Fanuc KAREL source: IO0221.KL

-- PROVISIONAL review KL for V1013-1; original PC SHA256 55de212278e1739486ba962373558651f202fb49e40d7032ca4ff645f1fc8ad3
-- Incomplete behavior may be omitted. Consult companion uncertainty JSON. Do not deploy.
PROGRAM IO0221
%NOLOCKGROUP
-- UNRESOLVED_LOCAL_POOL 5 cells at code offset 13; source declarations unknown
-- DIRECT_LOCAL_WORD_ACCESS alone does not prove INTEGER, REAL, or BOOLEAN
BEGIN
  -- UNRESOLVED_PC offsets 0-18; opcodes 2B,2C,7B
  -- UNRESOLVED_PC offsets 23-30; opcodes 9D,23
  -- UNRESOLVED_PC offsets 35-49; opcodes 2E,22,9D,33,35
  -- UNRESOLVED_PC offsets 54-61; opcodes 9D,23
  -- UNRESOLVED_PC offsets 66-77; opcodes 2E,23
  -- UNRESOLVED_PC offsets 82-133; opcodes 27,22,27,3F,27,3F,22,22,AF
  -- UNRESOLVED_PC offsets 138-142; opcodes 7F
  -- UNRESOLVED_PC offsets 147-151; opcodes 27,AA
  -- UNRESOLVED_PC offsets 156-160; opcodes 7F
END IO0221
